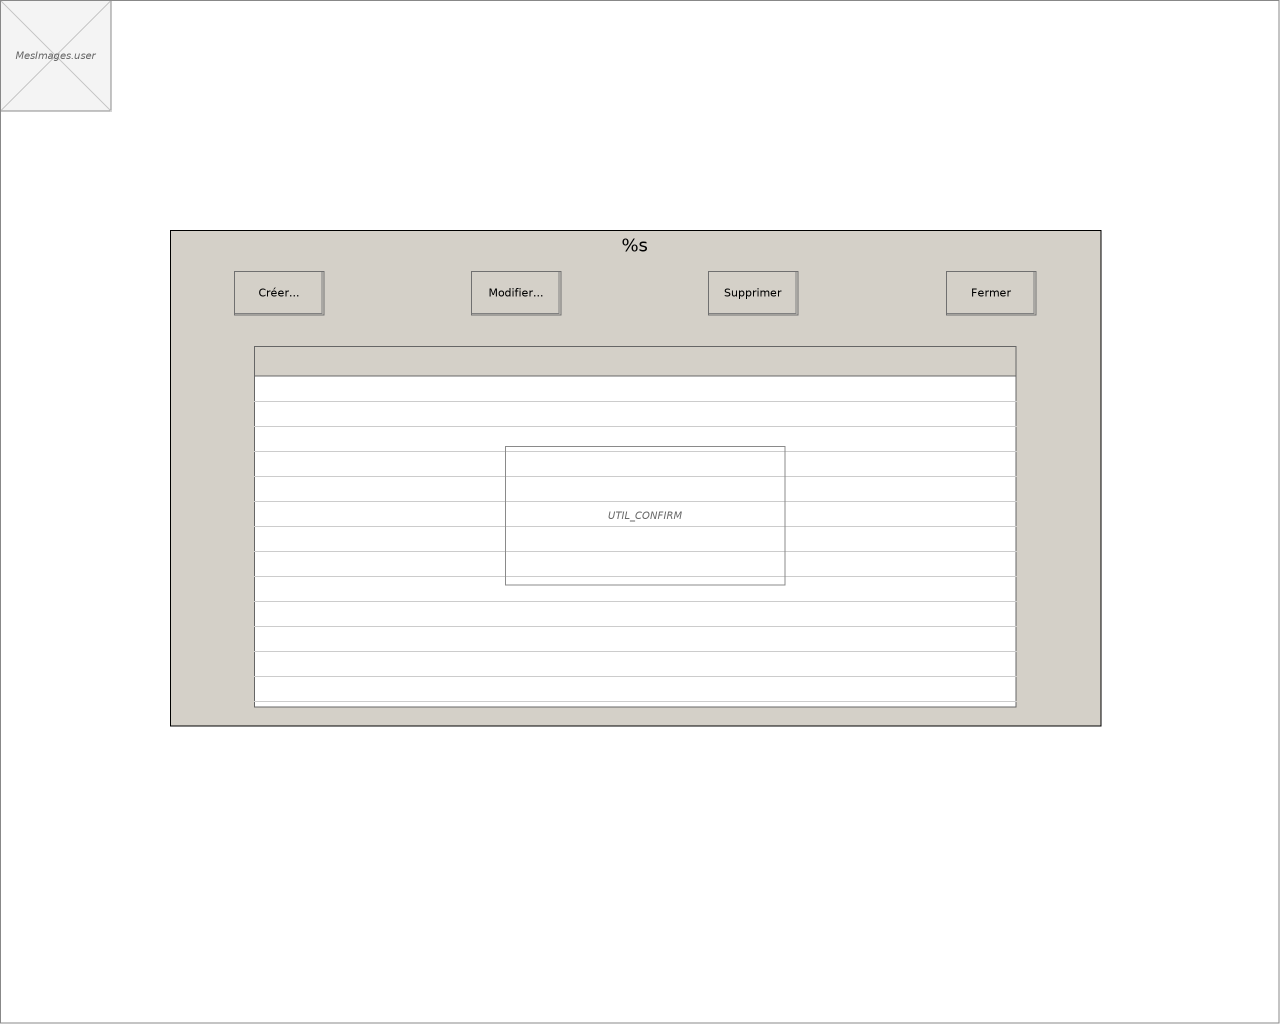
VISUALIZATION UTIL_GROUP  // 1280x1024
    RoundedRectangle (170,230 931x496)
    Image (0,0 111x111), image: MesImages.user
    Table (254,346 762x361), data array: PRG_USER.TBL_GROUP
        p1137915858: PRG_USER.LIGNE_GROUP
        p3854506369: PRG_USER.TBL_GROUP[INDEX].NOM
        p1892666644: PRG_USER.TBL_GROUP[INDEX].PROGRAMMATION
        p338671338: PRG_USER.TBL_GROUP[INDEX].MAINTENANCE
        p2170511999: PRG_USER.TBL_GROUP[INDEX].SUPERVISEUR
        p3723444502: PRG_USER.TBL_GROUP[INDEX].PRODUCTION
        p1218418051: PRG_USER.TBL_GROUP[INDEX].CONF_MACHINE
        p746581629: PRG_USER.TBL_GROUP[INDEX].FONCTION_SA
        p3104783080: PRG_USER.TBL_GROUP[INDEX].CONF_TRF
        p2501879983: PRG_USER.TBL_GROUP[INDEX].MODIF_ENLIGNE
        p7306298: PRG_USER.TBL_GROUP[INDEX].ARCHIVE_EV
        p1933151965: PRG_USER.TBL_GROUP[INDEX].DECONSIGNATION
        p2232123230: Nom du groupe
        p511219082: Pro. Ed
        p1755163831: Maint.
        p4092479075: Superv.
        p2237128397: Prod.
        p505689113: Conf.
        p1757482276: FoncSA.
    Textfield (231,233 808x25), "%s", text list: 'TextList_Util_Userlist', text index: 5
    Button (234,271 90x44), "Créer...", invisible if: PRG_USER.STOP_GROUP
        toggle PRG_USER.DD_EFFACE_NEW2
        OnMouseClick: change screen: UTIL_NEW_GROUP
    Button (471,271 90x44), "Modifier...", input disabled if: NOT PRG_USER.AUT_MOD_GRP
        toggle PRG_USER.DD_mod_group1
        OnMouseClick: change screen: UTIL_MOD_GROUP
    Button (708,271 90x44), "Supprimer", input disabled if: NOT PRG_USER.AUT_MOD_GRP
        toggle PRG_USER.VISU_FEN4
    Button (946,271 90x44), "Fermer", input disabled if: PRG_USER.VISU_FEN4
        OnMouseClick: change screen: UTIL_MENU
    Frame (505,446 280x139), invisible if: NOT PRG_USER.VISU_FEN4
        shows UTIL_CONFIRM(Num_Text := 19, OrdreDD := PRG_USER.DD_DEL_GROUP, Visu := PRG_USER.VISU_FEN4)
END_VISUALIZATION

(* stored: Version 1.1.0.1, ProductVersion 3.1.4024.10
   Visu UTIL_GROUP: Id {1fb5cdbc-a1b9-4d24-a3b4-2980581641d8} *)
